// TIA Portal V17 export
// export: Created 2025-03-05T08:02:53.9466706Z, ExportSetting WithDefaults, DisplayName Totally Integrated Automation Portal, DisplayVersion V17 Update 8, DisplayName TIA Portal Openness, DisplayVersion V17 Update 8, DisplayName TIA Portal Version Control Interface, DisplayVersion V17, DisplayName SINAMICS Startdrive Advanced, DisplayVersion V17 SP2, DisplayName SINAMICS Startdrive G110M, G120, G120C, G120D, G120P, G115D, DisplayVersion V17 SP2, DisplayName SINAMICS Startdrive G130, G150, S120, S150, SINAMICS MV, S210, DisplayVersion V17 SP2, DisplayName STEP 7 Professional, DisplayVersion V17 Update 8, DisplayName SINUMERIK ONE STEP 7 Toolbox, DisplayVersion V17 Update 12, DisplayName SINUMERIK 840D sl STEP 7 Toolbox, DisplayVersion V17 Update 12, DisplayName STEP 7 Safety, DisplayVersion V17 Update 6, DisplayName WinCC Advanced, DisplayVersion V17 Update 8
DATA_BLOCK "DB7252_FEEDER_2_UNIT_02_LINE_2"   // DB7252
{ DB_Accessible_From_OPC_UA := 'FALSE' }
VERSION : 0.1
// stored: AutoNumber false, DBAccessibleFromOPCUA false, DBAccessibleFromWebserver true, InstanceOfName FB7238_VARIABLES_PLC_HMI_FEEDERS, InstanceOfType FB
"FB7238_VARIABLES_PLC_HMI_FEEDERS"
   // VAR_INPUT
   //    GAS_FLOW_RATE_ACTUAL { ExternalAccessible := 'False'; ExternalVisible := 'False'; ExternalWritable := 'False'} : Real := 0.0;
   //    GAS_FLOW_RATE_AUTO { ExternalAccessible := 'False'; ExternalVisible := 'False'; ExternalWritable := 'False'} : Real := 0.0;
   //    DISC_SPEED_ACTUAL { ExternalAccessible := 'False'; ExternalVisible := 'False'; ExternalWritable := 'False'} : Real := 0.0;
   //    DISC_SPEED_AUTO { ExternalAccessible := 'False'; ExternalVisible := 'False'; ExternalWritable := 'False'} : Real := 0.0;
   //    STIRRER_SPEED_ACTUAL { ExternalAccessible := 'False'; ExternalVisible := 'False'; ExternalWritable := 'False'} : Real := 0.0;
   //    STIRRER_SPEED_AUTO { ExternalAccessible := 'False'; ExternalVisible := 'False'; ExternalWritable := 'False'} : Real := 0.0;
   //    HOPPER_TEMP_ACTUAL { ExternalAccessible := 'False'; ExternalVisible := 'False'; ExternalWritable := 'False'} : Real := 15.1;
   //    HOPPER_TEMP_AUTO { ExternalAccessible := 'False'; ExternalVisible := 'False'; ExternalWritable := 'False'} : Real := 0.0;
   //    HEATER_STATUS { ExternalAccessible := 'False'; ExternalVisible := 'False'; ExternalWritable := 'False'} : Byte := 0;
   //    HOPPER_STATUS { ExternalAccessible := 'False'; ExternalVisible := 'False'; ExternalWritable := 'False'} : Byte := 16#00;
   //    SELECTED_GAS : Int := 0;
   // END_VAR
   // VAR_OUTPUT
   //    HEATER_ON { ExternalAccessible := 'False'; ExternalVisible := 'False'; ExternalWritable := 'False'} : Bool := FALSE;
   //    HOPPER_ON { ExternalAccessible := 'False'; ExternalVisible := 'False'; ExternalWritable := 'False'} : Bool := FALSE;
   //    DISC_SPEED_WARN_UP_LIMIT { ExternalAccessible := 'False'; ExternalVisible := 'False'; ExternalWritable := 'False'} : Real := 10.0;
   //    DISC_SPEED_ALRM_UP_LIMIT { ExternalAccessible := 'False'; ExternalVisible := 'False'; ExternalWritable := 'False'} : Real := 2.0;
   //    DISC_SPEED_WARN_LOW_LIMIT { ExternalAccessible := 'False'; ExternalVisible := 'False'; ExternalWritable := 'False'} : Real := 15.0;
   //    DISC_SPEED_ALRM_LOW_LIMIT { ExternalAccessible := 'False'; ExternalVisible := 'False'; ExternalWritable := 'False'} : Real := 2.0;
   //    GAS_FLOW_RATE_WARN_UP_LIMIT { ExternalAccessible := 'False'; ExternalVisible := 'False'; ExternalWritable := 'False'} : Real := 3.0;
   //    GAS_FLOW_RATE_ALRM_UP_LIMIT { ExternalAccessible := 'False'; ExternalVisible := 'False'; ExternalWritable := 'False'} : Real := 4.0;
   //    GAS_FLOW_RATE_WARN_LOW_LIMIT { ExternalAccessible := 'False'; ExternalVisible := 'False'; ExternalWritable := 'False'} : Real := 15.0;
   //    GAS_FLOW_RATE_ALRM_LOW_LIMIT { ExternalAccessible := 'False'; ExternalVisible := 'False'; ExternalWritable := 'False'} : Real := 4.0;
   //    STIRRER_SPEED_WARN_UP_LIMIT { ExternalAccessible := 'False'; ExternalVisible := 'False'; ExternalWritable := 'False'} : Real := 10.0;
   //    STIRRER_SPEED_ALRM_UP_LIMIT { ExternalAccessible := 'False'; ExternalVisible := 'False'; ExternalWritable := 'False'} : Real := 5.0;
   //    STIRRER_SPEED_WARN_LOW_LIMIT { ExternalAccessible := 'False'; ExternalVisible := 'False'; ExternalWritable := 'False'} : Real := 99.0;
   //    STIRRER_SPEED_ALRM_LOW_LIMIT { ExternalAccessible := 'False'; ExternalVisible := 'False'; ExternalWritable := 'False'} : Real := 10.0;
   //    TEMP_ALRM_UP_LIMIT { ExternalAccessible := 'False'; ExternalVisible := 'False'; ExternalWritable := 'False'} : Real := 3.0;
   //    HOPPER_TEMP_MANUAL { ExternalAccessible := 'False'; ExternalVisible := 'False'; ExternalWritable := 'False'} : Real := 0.0;
   //    STIRRER_SPEED_MANUAL { ExternalAccessible := 'False'; ExternalVisible := 'False'; ExternalWritable := 'False'} : Real := 30.0;
   //    DISC_SPEED_MANUAL { ExternalAccessible := 'False'; ExternalVisible := 'False'; ExternalWritable := 'False'} : Real := 40.0;
   //    GAS_FLOW_RATE_MANUAL { ExternalAccessible := 'False'; ExternalVisible := 'False'; ExternalWritable := 'False'} : Real := 14.0;
   //    HOPPER_ON_REQ : Bool := FALSE;
   //    HOPPER_OFF_REQ : Bool := FALSE;
   //    HEATER_ON_REQ : Bool := FALSE;
   //    HEATER_OFF_REQ : Bool := FALSE;
   //    START_SEQUENCE_GAS_STEPS { ExternalAccessible := 'False'; ExternalVisible := 'False'; ExternalWritable := 'False'} : Int := 5;
   //    START_SEQUENCE_DISK_STEPS { ExternalAccessible := 'False'; ExternalVisible := 'False'; ExternalWritable := 'False'} : Int := 5;
   //    STOP_SEQUENCE_GAS_STEPS { ExternalAccessible := 'False'; ExternalVisible := 'False'; ExternalWritable := 'False'} : Int := 10;
   //    STOP_SEQUENCE_DISK_STEP { ExternalAccessible := 'False'; ExternalVisible := 'False'; ExternalWritable := 'False'} : Int := 10;
   //    STOP_SEQUENCE_PAUSE_STEP { ExternalAccessible := 'False'; ExternalVisible := 'False'; ExternalWritable := 'False'} : Int := 5;
   //    SELECTED_ARGON_GAS : Bool := TRUE;
   //    SELECTED_NITROGEN_GAS : Bool := FALSE;
   //    SELECTED_HELIUM_GAS : Bool;
   //    SELECTED_ARGON30_GAS : Bool;
   // END_VAR
   // VAR_IN_OUT
   //    FEEDER_LINE_OUT : "UDT_Feeder Line";
   // END_VAR
BEGIN
END_DATA_BLOCK
